FUNCTION_BLOCK E_BLINK (* Simulates a blinking signal (turning on and off for specific durations) *)
  (* Standard: 61499-1; Description: Copyright (c) 2025 HR Agrartechnik GmbH This program and the accompanying materials are made available under the terms of the Eclipse Public License 2.0 which is available at https://www.eclipse.org/legal/epl-2.0/ SPDX-License-Identifier: EPL-2.0 was a little inspired by this FUNCTION_BLOCK BLINK: https://content.helpme-codesys.com/en/libs/Util/Current/Signals/BLINK.html BUT while CODESYS keeps the last State, this FB return to FALSE on STOP. *)
  (* Version 1.0, 2025-02-15, Franz H??pfinger, HR Agrartechnik GmbH, initial API and implementation and/or initial documentation *)
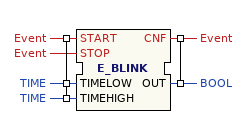
  EVENT_INPUT
    START WITH TIMELOW, TIMEHIGH; (* Start the perodic generation of events *)
    STOP; (* Stop the generation of events *)
  END_EVENT
  EVENT_OUTPUT
    CNF WITH OUT; (* Execution Confirmation *)
  END_EVENT
  VAR_INPUT
    TIMELOW : TIME; (* Time for OUT to be FALSE *)
    TIMEHIGH : TIME; (* Time for OUT to be TRUE *)
  END_VAR
  VAR_OUTPUT
    OUT : BOOL; (* Output value, starts with FALSE and switches between TRUE and FALSE for the given high and low times *)
  END_VAR
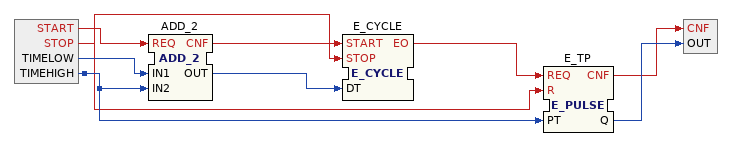
  FBS
    E_TP : E_PULSE;
    E_CYCLE : E_CYCLE;
    ADD_2 : ADD_2;
  END_FBS
  EVENT_CONNECTIONS
    E_CYCLE.EO TO E_TP.REQ;
    START TO ADD_2.REQ;
    ADD_2.CNF TO E_CYCLE.START;
    STOP TO E_CYCLE.STOP;
    E_TP.CNF TO CNF;
    STOP TO E_TP.R;
  END_CONNECTIONS
  DATA_CONNECTIONS
    ADD_2.OUT TO E_CYCLE.DT;
    TIMELOW TO ADD_2.IN1;
    TIMEHIGH TO ADD_2.IN2;
    E_TP.Q TO OUT;
    TIMEHIGH TO E_TP.PT;
  END_CONNECTIONS
END_FUNCTION_BLOCK
